// TIA Portal V19 export
FUNCTION_BLOCK "Main_Safety_RTG1"   // FB67, F_FBD
TITLE = Main_Safety_RTG1
AUTHOR : Siemens AG DI FA SUP
// stored: Namespace Safety
   VAR
      status { ExternalAccessible := 'False'; ExternalVisible := 'False'; ExternalWritable := 'False'} : "Safety.typeDataFromSafety";
      statAck { ExternalWritable := 'False'} : Bool;   // Signal Bit for acknowledgement
      instAckOP { ExternalWritable := 'False'} : ACK_OP;   // Acknowledge command from the HMI
      instAckGL { ExternalWritable := 'False'} : ACK_GL;   // Global acknowledgement for all F-I/Os in the F-runtime group
      instSafetyZone1Actuators { ExternalWritable := 'False'} : "Safety.SafetyZone1Actuators";
      instLSafeEStopDrvZone1 { ExternalWritable := 'False'} : "Safety.LSafe_EStopDrives";
      instLSafeFDoorDrvZone1 { ExternalWritable := 'False'} : "Safety.LSafe_FDoorDrives";
      instStatusSummary { ExternalWritable := 'False'} : "Safety.StatusSummary";
   END_VAR
   VAR_TEMP
      tempAckHMI : Bool;   // Temp Signal for Acknowledgement from HMI
      tempEStopE0 : Bool;   // Temp State of EStop E0
      tempEStopE1 : Bool;   // Temp State of EStop E1
      tempFDoorRFID : Bool;   // Temp State of 3SE63 RFID protective door switch
      tempVSFDoorRFID : Bool;   // Temp Value State of 3SE63 RFID protective door switch
      tempRelEStopZone1STO : Bool;   // Temp STO release signal from Estop Function Zone 1
      tempRelFDoorZone1STO : Bool;   // Temp STO release signal from FDoor Function Zone 1
      tempAckReqActuatorsZone1 : Bool;   // Temp Acknowledge request Actuators Zone 1
      tempSTOActiveZone1 : Bool;   // Temp STO active Zone 1
   END_VAR
   VAR CONSTANT
      ALWAYS_FALSE : Bool;   // Const false
      ALWAYS_TRUE : Bool := true;   // Const true
   END_VAR
BEGIN

REGION Network 1: Acknowledgement
   // This network contains the acknowledgement for the safety-program.
   // Safety could be acknowledge by the HMI or by reset buttons connected to the units.
   // Ack_OP enables fail-safe acknowledgement from an operator control and monitoring system. 
   // Ack_GL reintegrates all passivated F-I/O modules of the calling F-Runtime group.
   // In the basic AF, no reset buttons in the units are connected, so
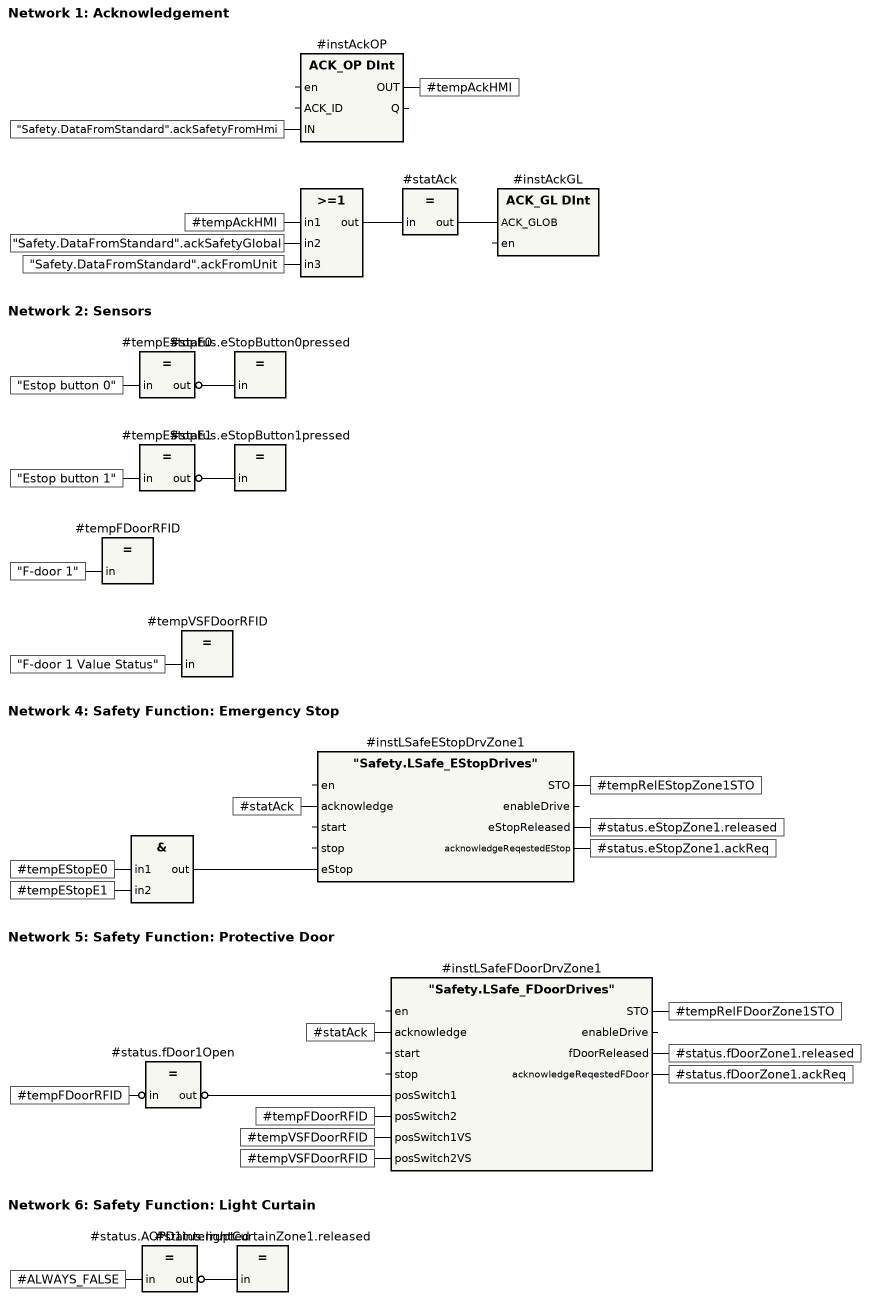
   #instAckOP(IN := "Safety.DataFromStandard".ackSafetyFromHmi, OUT => #tempAckHMI);   // ACK_OP
   #statAck := #tempAckHMI OR "Safety.DataFromStandard".ackSafetyGlobal OR "Safety.DataFromStandard".ackFromUnit;
   #instAckGL(ACK_GLOB := #statAck);   // ACK_GL
END_REGION

REGION Network 2: Sensors
   // Copy input tags from failsafe-input modules.
   #tempEStopE0 := "Estop button 0";
   #status.eStopButton0pressed := NOT "Estop button 0";
   #tempEStopE1 := "Estop button 1";
   #status.eStopButton1pressed := NOT "Estop button 1";
   #tempFDoorRFID := "F-door 1";
   #tempVSFDoorRFID := "F-door 1 Value Status";
END_REGION

REGION Network 3: ********** Safety Zone 1 **********
END_REGION

REGION Network 4: Safety Function: Emergency Stop
   // *** Safety Zone 1 - Safety Function: Emergency Stop***
   // This function implements a safe shutdown (STO) of drives in emergency. 
   // When the emergency button is pressed, the actuator(s) are switched off with STO.
   // For more information, please refer to:  https://support.industry.siemens.com/cs/ww/en/view/109793462
   #instLSafeEStopDrvZone1(acknowledge := #statAck,   // "Safety.LSafe_EStopDrives"
                           eStop := #tempEStopE0 AND #tempEStopE1,
                           STO => #tempRelEStopZone1STO,
                           eStopReleased => #status.eStopZone1.released,
                           acknowledgeReqestedEStop => #status.eStopZone1.ackReq);
END_REGION

REGION Network 5: Safety Function: Protective Door
   // *** Safety Zone 1 - Safety Function: Protective Door ***
   // This function implements safe protective door monitoring without guard looking.
   // The actuator(s) are switched off (STO) safely when the protective door is opend during operation or a fault is detected.
   // For more information, please refer to:  https://support.industry.siemens.com/cs/ww/en/view/109793462
   #status.fDoor1Open := NOT #tempFDoorRFID;
   #instLSafeFDoorDrvZone1(acknowledge := #statAck,   // "Safety.LSafe_FDoorDrives"
                           posSwitch1 := NOT (NOT #tempFDoorRFID),
                           posSwitch2 := #tempFDoorRFID,
                           posSwitch1VS := #tempVSFDoorRFID,
                           posSwitch2VS := #tempVSFDoorRFID,
                           STO => #tempRelFDoorZone1STO,
                           fDoorReleased => #status.fDoorZone1.released,
                           acknowledgeReqestedFDoor => #status.fDoorZone1.ackReq);
END_REGION

REGION Network 6: Safety Function: Light Curtain
   // *** Safety Zone 1 - Safety Function: Light Curtain ***
   // This function is not implemented. Additionally required safety functions can be implemented in accordance to the risk assessment. Application examples to commonly used safety functions can be found in SIOS and selected via Safety Select: https://support.industry.siemens.com/cs/ww/en/view/109773295
   #status.AOPD1interrupted := #ALWAYS_FALSE;
   #status.lightCurtainZone1.released := NOT #ALWAYS_FALSE;
END_REGION

REGION Network 7: Actuators
   // *** Safety Zone 1 - Actuators ***
   // This network implements the interconnection to the actuator hardware. 
   // The Safety integrated functions of drives 1 to 6 are controlled via PROFIsafe with LDrvSafe function blocks.
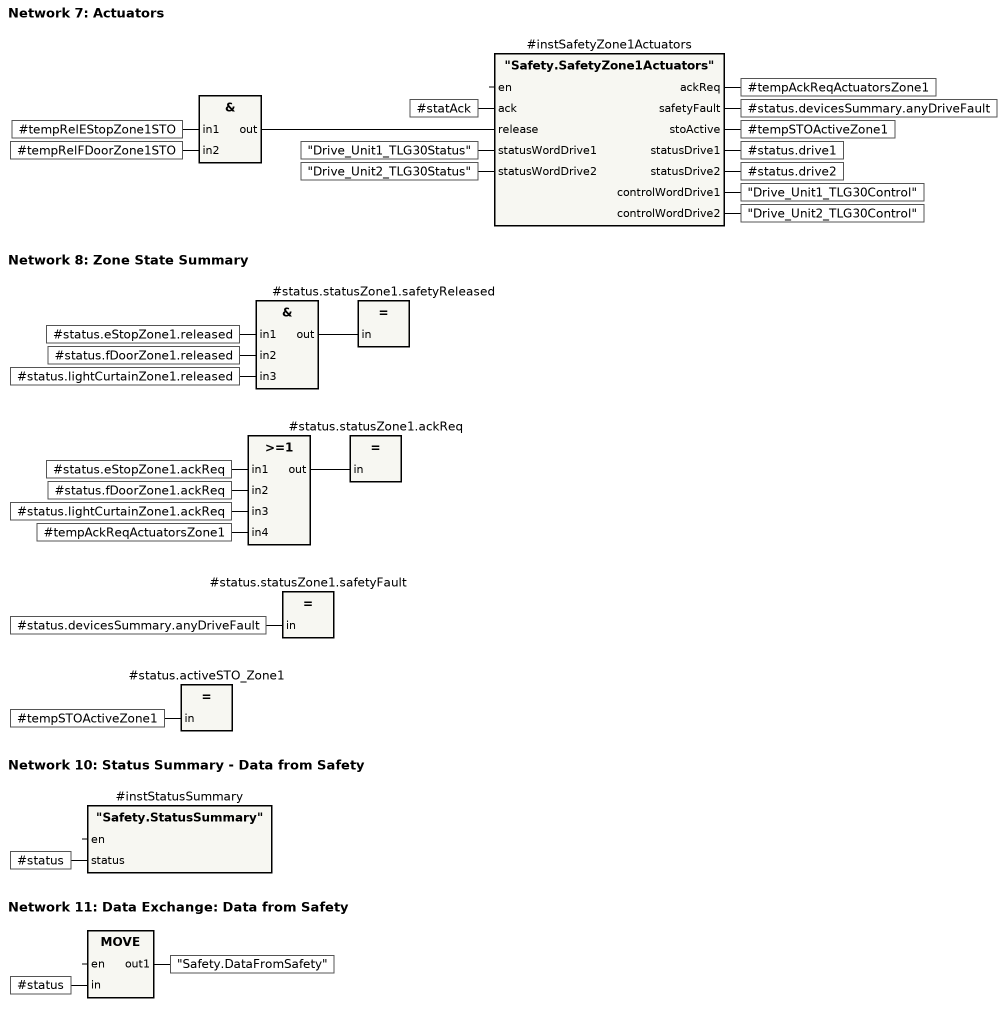
   #instSafetyZone1Actuators(ack := #statAck,   // "Safety.SafetyZone1Actuators"
                           release := #tempRelEStopZone1STO AND #tempRelFDoorZone1STO,
                           statusWordDrive1 := "Drive_Unit1_TLG30Status",
                           statusWordDrive2 := "Drive_Unit2_TLG30Status",
                           ackReq => #tempAckReqActuatorsZone1,
                           safetyFault => #status.devicesSummary.anyDriveFault,
                           stoActive => #tempSTOActiveZone1,
                           statusDrive1 => #status.drive1,
                           statusDrive2 => #status.drive2,
                           controlWordDrive1 => "Drive_Unit1_TLG30Control",
                           controlWordDrive2 => "Drive_Unit2_TLG30Control");
END_REGION

REGION Network 8: Zone State Summary
   // *** Safety Zone 1 - Zone State Summary ***
   // This network summerizes the states of the safety functions for diagnostics in the standard user program.
   #status.statusZone1.safetyReleased := #status.eStopZone1.released AND #status.fDoorZone1.released AND #status.lightCurtainZone1.released;
   #status.statusZone1.ackReq := #status.eStopZone1.ackReq OR #status.fDoorZone1.ackReq OR #status.lightCurtainZone1.ackReq OR #tempAckReqActuatorsZone1;
   #status.statusZone1.safetyFault := #status.devicesSummary.anyDriveFault;
   #status.activeSTO_Zone1 := #tempSTOActiveZone1;
END_REGION

REGION Network 9: *************************************
END_REGION

REGION Network 10: Status Summary - Data from Safety
   // Summarize the Status Information from all Safety Zones and form general diagnostic bits.
   #instStatusSummary(status := #status);   // "Safety.StatusSummary"
END_REGION

REGION Network 11: Data Exchange: Data from Safety
   // Move temporary status information to data exchange DB "DataFromSafety"
   "Safety.DataFromSafety" := #status;
END_REGION
END_FUNCTION_BLOCK
